TYPE ST_Value :
STRUCT
	Setpoint	: REAL;
	Actual		: REAL;
END_STRUCT
END_TYPE

(* stored: Version 1.1.0.1, ProductVersion 3.1.4024.14
   DUT ST_Value: Id {d70f96fe-38ae-08cb-207b-f1433e0b6228} *)
